{attribute 'GeneratedUsingTerminal: EL3356-0000-0017'}
{attribute addProperty BoxType "EL3356-0000-0017"}
{attribute addProperty Id "Start_calibrationBOOL1Disable_calibrationBOOL1Input_freezeBOOL1TaraBOOL1"}
{attribute addProperty CRC "2933667662"}
{attribute addProperty Size "4"}
TYPE Ctrl_AEDC374E :
STRUCT
	{attribute addProperty Name "Start_calibration"}
	Start_calibration : BOOL;
	{attribute addProperty Name "Disable_calibration"}
	Disable_calibration : BOOL;
	{attribute addProperty Name "Input_freeze"}
	Input_freeze : BOOL;
	{attribute addProperty Name "Tara"}
	Tara : BOOL;
END_STRUCT
END_TYPE

(* stored: Version 1.2.0.0, ProductVersion 3.1.4024.9
   DUT Ctrl_AEDC374E: Id {56b94e35-ed8b-4016-966b-cc2ec3295985} *)
